// SIMATIC S7-200 project (STEP 7-Micro/WIN), CPU 226 CN REL 02.01

SYMBOL_TABLE 用户定义1
速度接收脉冲           I0.0
变频器故障            I0.1
启动               I0.2
停止               I0.3
手动自动             I0.4
模式1模式2           I0.5
皮带上升下降           I0.6
皮带转动             I0.7
滚筒正转             I1.0
滚筒反转             I1.1
皮带减速信号1          I1.2
皮带减速信号2          I1.3
皮带停止信号           I1.4
左出信号1            I1.5
左出信号2            I1.6
右出信号1            I1.7
右出信号2            I2.0
辊台减速信号           I2.1
辊台停止信号           I2.2
打孔机允许送板信号        I2.3
打孔机运行信号          I2.4
紧急停止             I2.5
速度输出脉冲           Q0.0
运行指示灯            Q0.1
下料齐板             Q0.2
上料齐板             Q0.3
皮带升降汽缸           Q0.4
下料挡板             Q0.5
允许双端铣送板          Q0.6
允许悬臂机送板          Q0.7
上下料机模式输出         Q1.0
给打孔机脉冲信号         Q1.1
给上下料机械手运行信号      Q1.2
给双端铣运行信号         Q1.3
异常指示             Q1.7
END_SYMBOL_TABLE

ORGANIZATION_BLOCK 主程序:OB1
TITLE=~~~~~PLC程序实例~~~~~
// 程序注释
// 系统启动时，运行初始化程序，将皮带速度变量、滚筒1速度变量和滚筒2速度变量设置为默认值，同时初始化其他相关变量并设置内部状态。操作员通过启动按钮启动系统，但需处于自动模式且变频器无故障，同时满足其他内部条件。在手动模式下，操作员可通过皮带上升下降按钮控制皮带升降气缸，或使用滚筒正转和反转按钮调整滚筒速度，并确保正反转不会同时发生。
// 进入自动模式后，模式切换开关决定运行模式。在模式1（双端铣加工）下，皮带升降气缸抬起皮带，皮带速度驱动板材移动，随后系统等待皮带停止和到位信号未触发时，通知双端铣接收板材。接着，若打孔机准备就绪，发出脉冲信号，根据方向选择向左或向右输送板材。在模式2（悬臂机加工）下，下料挡板打开，随后在辊台停止时通知悬臂机取板，同时滚筒速度驱动板材移动。
// 系统运行状态通过运行指示灯显示，异常指示灯在变频器无故障时亮起。若按下紧急停止按钮，部分输出如皮带升降气缸和脉冲信号立即复位，确保安全停止。
// 
BEGIN
Network 1 // 

LD     SM0.1
CALL   初始化程序:SBR0
?000
?000
Network 2
LD     SM0.1
MOVB   1, VB19
MOVW   16#1, VW20
MOVW   +0, VW22
MOVW   16#1, VW24
MOVW   +0, VW26
MOVW   16#1, VW28
MOVW   +0, VW30
S      M2.6, 1
Network 4
LDN    M2.1
LPS
AB=    VB19, 1
LPS
MOVB   16#1, VB11
AN     M2.6
MOVW   16#2000, VW13
LPP
AN     M2.6
MOVW   VW20, VW15
LPP
AB=    VB19, 2
LPS
AN     M2.6
MOVW   16#2001, VW13
LPP
AN     M2.6
MOVW   VW22, VW15
Network 5
LDN    M2.1
LPS
AB=    VB19, 3
LPS
MOVB   16#2, VB11
AN     M2.6
MOVW   16#2000, VW13
LPP
AN     M2.6
MOVW   VW24, VW15
LPP
AB=    VB19, 4
LPS
AN     M2.6
MOVW   16#2001, VW13
LPP
AN     M2.6
MOVW   VW26, VW15
Network 6
LDN    M2.1
LPS
AB=    VB19, 5
LPS
MOVB   16#3, VB11
AN     M2.6
MOVW   16#2000, VW13
LPP
AN     M2.6
MOVW   VW28, VW15
LRD
AB=    VB19, 6
LPS
AN     M2.6
MOVW   16#2001, VW13
LPP
AN     M2.6
MOVW   VW30, VW15
LPP
A      M2.6
MOVW   16#2002, VW13
MOVW   16#2, VW15
Network 8
LD     SM0.0
AN     M2.4
TON    T38, +40
Network 9
LD     T38
O      M2.4
LPS
=      M2.4
A      M2.6
TON    T39, 30
LPP
A      T39
R      M2.6, 1
Network 10
LD     M2.4
LPS
AN     M2.5
TON    T34, +2
LRD
A      T34
=      M2.5
LPP
A      M2.5
LPS
AN     M2.2
S      M2.1, 1
LPP
A      M2.2
R      M2.1, 1
Network 11
LD     M2.1
=      M2.2
Network 12
// 发送命令模块程序
LD     M2.1
EU
LPS
CALL   CRC校验程序:SBR2
AB<    VB19, 7
INCB   VB19
LRD
AB=    VB19, 7
MOVB   1, VB19
LRD
S      M2.0, 1
LPP
R      M10.0, 1
Network 14
LD     M2.0
EU
XMT    VB10, 1
Network 15
LD     SM4.6
EU
R      M2.0, 1
Network 17
// 双端洗速度检测
LDN    M2.7
TOF    T32, +500
Network 18
LD     T32
=      M2.7
Network 19
// 手动部分程序
// 
LDN    M20.0
AN     手动自动:I0.4
MOVW   5000, VW22
MOVW   5000, VW26
MOVW   5000, VW30
Network 20
LDN    M20.0
AN     手动自动:I0.4
A      皮带上升下降:I0.6
EU
LPS
AN     M3.0
S      皮带升降汽缸:Q0.4, 1
LPP
A      M3.0
R      皮带升降汽缸:Q0.4, 1
Network 21
LD     皮带升降汽缸:Q0.4
=      M3.0
Network 22
LDN    M20.0
AN     手动自动:I0.4
A      皮带转动:I0.7
LPS
EU
MOVW   16#12, VW20
LPP
ED
MOVW   +1, VW20
Network 23
LDN    M20.0
AN     手动自动:I0.4
A      滚筒正转:I1.0
LPS
EU
AN     滚筒反转:I1.1
MOVW   16#12, VW24
MOVW   16#12, VW28
LPP
ED
MOVW   +1, VW24
MOVW   +1, VW28
Network 24
LDN    M20.0
AN     手动自动:I0.4
A      滚筒反转:I1.1
LPS
EU
AN     滚筒正转:I1.0
MOVW   16#22, VW24
MOVW   16#22, VW28
LPP
ED
MOVW   +1, VW24
MOVW   +1, VW28
Network 25
// 自动程序
LD     M2.4
AN     M2.6
A      变频器故障:I0.1
A      启动:I0.2
A      手动自动:I0.4
AN     M20.0
EU
S      M20.0, 1
Network 26
LDN    M20.1
AN     M20.2
A      M20.0
LPS
AN     模式1模式2:I0.5
EU
S      M20.1, 1
LPP
A      模式1模式2:I0.5
EU
S      M20.2, 1
Network 27
LD     M20.1
CALL   自动模式1:SBR1
=      上下料机模式输出:Q1.0
=      给双端铣运行信号:Q1.3
Network 28
LD     M20.2
CALL   自动模式2:SBR3
Network 29
LD     M20.1
O      M20.2
=      给上下料机械手运行信号:Q1.2
Network 30
LD     M20.0
AN     手动自动:I0.4
EU
=      M20.4
Network 31
LD     手动自动:I0.4
AN     停止:I0.3
O      SM0.1
O      M20.4
ON     紧急停止:I2.5
R      M20.0, 3
R      M21.0, 8
R      M23.0, 8
R      皮带升降汽缸:Q0.4, 4
R      下料齐板:Q0.2, 2
R      给打孔机脉冲信号:Q1.1, 1
MOVW   16#1, VW20
MOVW   16#1, VW24
MOVW   16#1, VW28
Network 32
LD     M20.0
=      运行指示灯:Q0.1
Network 33
LD     M2.4
A      紧急停止:I2.5
EU
S      M2.6, 1
Network 34
LDN    变频器故障:I0.1
AN     M2.6
=      异常指示:Q1.7
END_ORGANIZATION_BLOCK

SUBROUTINE_BLOCK 初始化程序:SBR0
TITLE=子程序注释
BEGIN
Network 1
// \\初始化Prot1口，9600，8，1，E
LD     SM0.0
LPS
MOVB   16#C9, SMB130
AN     SM0.0
MOVB   16#C9, SMB30
LPP
MOVB   16#8, VB10
Network 2
// 高速计数器初始化
LD     SM0.0
MOVB   16#FC, SMB37
HDEF   0, 0
MOVD   +0, SMD38
MOVD   +500000, SMD42
HSC    0
Network 3
// 打开定时器中断
LD     SM0.0
ATCH   INT_0:INT0, 21
ENI
END_SUBROUTINE_BLOCK

SUBROUTINE_BLOCK 自动模式1:SBR1
TITLE=子程序注释
BEGIN
Network 1
// 双端铣输送带速度跟踪
LD     SM0.0
DTI    VD50, VW60
MOVW   VW60, VW64
*I     +60, VW64
AN     M22.0
MOVW   VW64, VW22
Network 2
LD     SM0.0
R      下料挡板:Q0.5, 1
Network 3
// 皮带上升，皮带启动
// 
LDN    M21.0
A      M20.1
LPS
AN     左出信号1:I1.5
AN     左出信号2:I1.6
AN     右出信号1:I1.7
AN     右出信号2:I2.0
S      皮带升降汽缸:Q0.4, 1
LRD
LD     左出信号1:I1.5
O      左出信号2:I1.6
O      右出信号1:I1.7
O      右出信号2:I2.0
ALD
S      M21.0, 3
LPP
LPS
MOVW   16#12, VW20
A      皮带升降汽缸:Q0.4
TON    T40, +10
LPP
A      T40
S      M21.0, 1
Network 4 // 网络标题
// 发出双端铣送板信号
// 
LDN    M21.1
A      M21.0
LPS
AN     皮带减速信号1:I1.2
AN     皮带减速信号2:I1.3
AN     皮带停止信号:I1.4
AN     左出信号1:I1.5
AN     左出信号2:I1.6
AN     右出信号1:I1.7
AN     右出信号2:I2.0
TON    T41, +10
LRD
LD     皮带减速信号1:I1.2
O      皮带减速信号2:I1.3
O      皮带停止信号:I1.4
ALD
AN     左出信号1:I1.5
AN     左出信号2:I1.6
AN     右出信号1:I1.7
AN     右出信号2:I2.0
S      M21.1, 1
LPP
A      T41
S      允许双端铣送板:Q0.6, 1
S      M21.1, 1
Network 5
// 皮带停止，皮带下降
LDN    M21.2
A      M21.1
LPS
A      皮带停止信号:I1.4
TON    T42, +4
LRD
LD     皮带减速信号1:I1.2
O      皮带减速信号1:I1.2
AN     M22.0
ALD
MOVW   +2000, VW22
R      允许双端铣送板:Q0.6, 1
S      M22.0, 1
LPP
A      T42
R      皮带升降汽缸:Q0.4, 1
MOVW   16#1, VW20
R      M22.0, 1
S      M21.2, 1
Network 6
// 左右方向选择
LDN    M21.3
AN     M21.4
A      M21.2
LPS
A      打孔机允许送板信号:I2.3
MOVW   16#22, VW24
MOVW   +5000, VW26
S      给打孔机脉冲信号:Q1.1, 1
S      M21.3, 1
LPP
AN     M21.5
AN     打孔机允许送板信号:I2.3
MOVW   16#12, VW24
MOVW   +5000, VW26
MOVW   16#12, VW28
MOVW   +5000, VW30
S      M21.4, 1
Network 7
// 向左送板
LD     M21.3
LPS
LD     左出信号1:I1.5
O      左出信号2:I1.6
ALD
AN     M22.1
S      M22.1, 1
LRD
AN     左出信号1:I1.5
AN     左出信号2:I1.6
A      M22.1
TON    T43, +20
LPP
A      T43
AN     皮带减速信号1:I1.2
AN     皮带减速信号2:I1.3
AN     皮带停止信号:I1.4
AN     左出信号1:I1.5
AN     左出信号2:I1.6
R      M21.0, 5
R      M22.1, 1
R      给打孔机脉冲信号:Q1.1, 1
MOVW   16#1, VW24
Network 8
// 向右送板
LD     M21.4
LPS
LD     右出信号1:I1.7
O      右出信号2:I2.0
ALD
AN     M22.2
S      M22.2, 1
LRD
AN     右出信号1:I1.7
AN     右出信号2:I2.0
A      M22.2
TON    T44, +20
LPP
A      T44
AN     左出信号1:I1.5
AN     左出信号2:I1.6
AN     右出信号1:I1.7
AN     右出信号2:I2.0
S      M21.5, 1
R      M21.0, 5
R      M22.2, 1
MOVW   16#1, VW24
Network 9
// 向右送板到位，发出允许取板信号
// 
LDN    M21.6
A      M21.5
LPS
A      辊台减速信号:I2.1
EU
MOVW   +2500, VW30
LPP
A      辊台停止信号:I2.2
TON    T45, +15
A      T45
MOVW   16#1, VW28
S      M21.6, 1
Network 10
LDN    M21.7
A      M21.6
LPS
EU
S      下料齐板:Q0.2, 1
LRD
A      下料齐板:Q0.2
TON    T46, 20
LPP
A      T46
S      允许悬臂机送板:Q0.7, 1
R      下料齐板:Q0.2, 1
S      M21.7, 1
Network 11
LD     M21.7
AN     辊台减速信号:I2.1
AN     辊台停止信号:I2.2
R      M21.5, 3
R      允许悬臂机送板:Q0.7, 1
END_SUBROUTINE_BLOCK

SUBROUTINE_BLOCK CRC校验程序:SBR2
TITLE=PROGRAM COMMENTS
BEGIN
Network 1 // Network Title
// Network Comment
LDN    M10.0
MOVW   16#FFFF, VW100
MOVB   16#6, VB12
MOVD   &VB11, VD0
Network 2
LDN    M10.0
FOR    VW6, +1, +6
Network 3
LD     SM0.0
XORB   *VD0, VB101
INCD   VD0
Network 4
LD     SM0.0
FOR    VW8, +1, +8
Network 5
LD     SM0.0
LPS
MOVW   16#1, VW102
ANDW   VW100, VW102
AW=    VW102, +1
SRW    VW100, 1
XORW   16#A001, VW100
LPP
AW=    VW102, +0
SRW    VW100, 1
Network 6
NEXT
Network 7
NEXT
Network 8
LD     SM0.0
S      M10.0, 1
Network 9
LD     SM0.0
MOVB   VB101, VB17
MOVB   VB100, VB18
Network 23 // 网络标题
// 网络注释
END_SUBROUTINE_BLOCK

SUBROUTINE_BLOCK 自动模式2:SBR3
TITLE=子程序注释
BEGIN
Network 1
LD     SM0.0
S      下料挡板:Q0.5, 1
R      皮带升降汽缸:Q0.4, 1
Network 2 // 网络标题
// 发出取板信号
LDN    M23.0
A      M20.2
LDN    辊台停止信号:I2.2
O      M23.5
ALD
S      允许悬臂机送板:Q0.7, 1
S      M23.0, 1
Network 3
// 辊台启动
LDN    M23.1
A      M23.0
A      辊台停止信号:I2.2
LPS
AN     上料齐板:Q0.3
TON    T50, +40
LRD
A      T50
S      上料齐板:Q0.3, 1
LRD
A      上料齐板:Q0.3
TON    T53, 20
LPP
A      T53
MOVW   16#22, VW24
MOVW   +5000, VW26
MOVW   16#22, VW28
MOVW   +5000, VW30
R      上料齐板:Q0.3, 1
R      M23.5, 1
R      允许悬臂机送板:Q0.7, 1
S      给打孔机脉冲信号:Q1.1, 1
S      M23.1, 1
Network 4
LDN    M23.2
A      M23.1
A      皮带停止信号:I1.4
EU
S      M23.2, 1
Network 5
// 待料，继续送板判断
LDN    M23.3
A      M23.2
LPS
A      打孔机允许送板信号:I2.3
S      M23.3, 1
S      给打孔机脉冲信号:Q1.1, 1
MOVW   16#22, VW24
MOVW   16#22, VW28
LPP
AN     打孔机允许送板信号:I2.3
MOVW   16#1, VW24
MOVW   16#1, VW28
R      给打孔机脉冲信号:Q1.1, 1
Network 6
LDN    M23.4
A      M23.3
LD     左出信号1:I1.5
O      左出信号2:I1.6
ALD
EU
S      M23.4, 1
Network 7
LD     M23.4
AN     皮带停止信号:I1.4
AN     左出信号1:I1.5
AN     左出信号2:I1.6
TON    T51, +20
A      T51
MOVW   16#1, VW24
MOVW   16#1, VW28
TON    T52, +10
A      T52
R      给打孔机脉冲信号:Q1.1, 1
S      M23.5, 1
R      M23.0, 5
END_SUBROUTINE_BLOCK

INTERRUPT_BLOCK INT_0:INT0
TITLE=中断程序注释
BEGIN
Network 1 // 网络标题
// 网络注释
LD     SM0.0
MOVW   +0, T32
MOVD   HC0, VD50
MOVB   16#C4, VB37
MOVD   +0, SMD38
HSC    0
INCD   VD54
END_INTERRUPT_BLOCK
